// TIA Portal V20 export
TYPE "LKinCtrl_typePathDynamics"
   STRUCT
      velocity : LReal := -1.0;   // >0.0: configured value used; <0.0: default TO setting used; for cmdType = 100 ==> waitTime in ms
      acceleration : LReal := -1.0;   // >0.0: configured value used; <0.0: default TO setting used
      deceleration : LReal := -1.0;   // >0.0: configured value used; <0.0: default TO setting used
      jerk : LReal := -1.0;   // >0.0: configured value used; <0.0: default TO setting used
   END_STRUCT;
END_TYPE
